// TIA Portal V16 export
// export: Created 2025-08-30T12:59:16.5989585Z, ExportSetting WithDefaults, DisplayName Totally Integrated Automation Portal, DisplayVersion V16, DisplayName TIA Portal Version Control Interface, DisplayVersion V16, DisplayName TIA Portal Openness, DisplayVersion V16, DisplayName STEP 7 Professional, DisplayVersion V16, DisplayName STEP 7 Safety, DisplayVersion V16, DisplayName WinCC Advanced, DisplayVersion V16
DATA_BLOCK "ProductCounter"   // DB21
// stored: AutoNumber true, InstanceOfName CTU_SFB, OfSystemLibElement CTU, OfSystemLibVersion 1.0
"CTU_SFB"
   // VAR_INPUT
   //    CU : Bool;
   //    R : Bool;
   //    PV : Int;
   // END_VAR
   // VAR_OUTPUT
   //    Q : Bool;
   //    CV : Int;
   // END_VAR
   // VAR RETAIN
   //    CUO : Bool;
   // END_VAR
BEGIN
END_DATA_BLOCK
